RoboDK station: Deployability.rdk

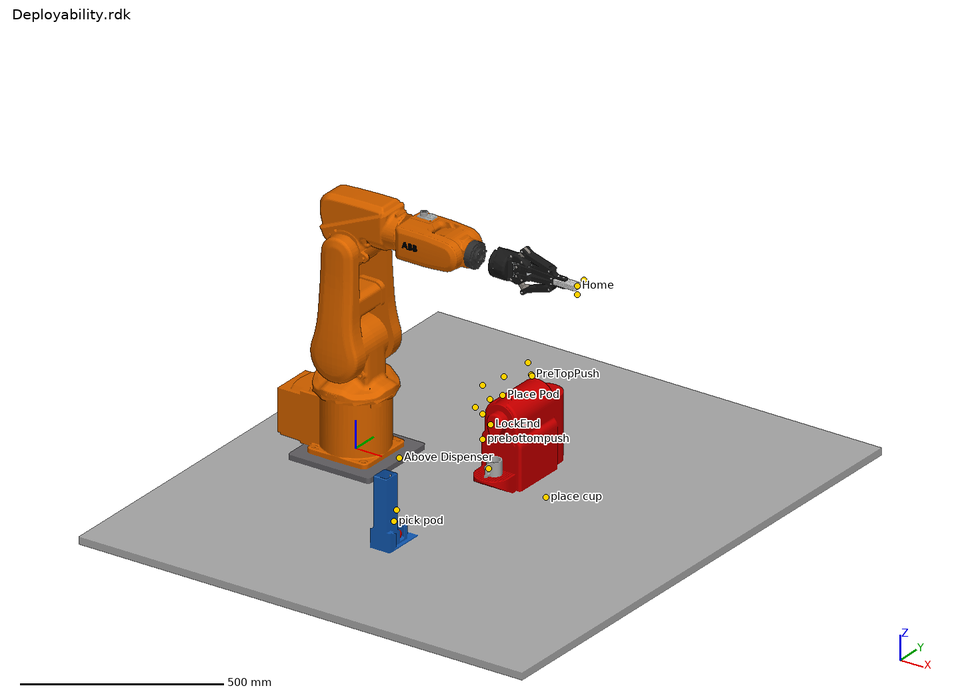
[picture v0: the station drawn from its stored meshes, robots at their saved joint values, targets as dots, program paths as lines]
Station Deployability (saved by RoboDK 5.6.7). Poses are relative to the parent item; angles as X-Y-Z fixed-axis rotations.
Station parameters (name, value as stored): LIN64
  - frame ABB IRB 120-3/0.6 Base at (-2.05, 0, 0) mm
    - target pick pod (Cartesian target) at (354.6, -342.93, 36.52) mm, rotated rx 177.2 ry -1.29 rz 4.29 deg; joints [-43.236, 48.573, -23.215, 1.337, 64.052, 131.893]
    - target Home (Cartesian target) at (664, 0, 630) mm, rotated rx 0 ry 90 rz 0 deg; joints [0, 0, 0, 0, 0, 0]
    - target Place Pod (Cartesian target) at (394.38, 64.87, 228.85) mm, rotated rx 178.74 ry -0.46 rz 90.36 deg; joints [16.786, 24.373, -22.849, 0.084, 87.136, 192.491]
    - target Above Dispenser (Cartesian target) at (372.26, -344.62, 215.16) mm, rotated rx -179.63 ry -1.29 rz 4.29 deg; joints [-43.653, 58.022, -72.664, 1.244, 104.052, 132.364]
    - robot ABB IRB 120-3/0.6: 6 axes, payload 3 kg, reach 580 mm, repeatability 0.01 mm, weight 25 kg
        modified DH rows (alpha deg, a mm, theta deg, d mm): 0, 0, 0, 290; -90, 0, -90, 0; 0, 270, 0, 0; -90, 70, 0, 302; 90, 0, 0, 0; -90, 0, 180, 72
        joint limits [-165, -110, -90, -160, -120, -400] to [165, 110, 70, 160, 120, 400]; home [0, 0, 0, 0, 0, 0]; saved at [-0.052, 0.172, -0.115, 0.095, 0.169, -0.086]
      - tool RobotiQ 2F-140 Gripper (Closed), TCP at (0, 0, 290) mm, size 124 x 75 x 244.3 mm
    - target PreTopPush (Cartesian target) at (397.09, 185.15, 238.21) mm, rotated rx -179.43 ry 2.35 rz -179.98 deg; joints [26.28, 27.432, -27.478, -1.552, 88.195, 26.292] of ABB IRB 120-3/0.6
    - target prebottompush (Cartesian target) at (368.51, 16.26, 120.96) mm, rotated rx 0 ry 90 rz 52.6 deg; joints [-61.285, 60.722, 28.546, -113.883, -90.297, 0.67] of ABB IRB 120-3/0.6
    - target PostTopPush (Cartesian target) at (396.91, -54.26, 245.05) mm, rotated rx -179.43 ry 2.35 rz -179.98 deg; joints [-7.551, 17.486, -15.446, -0.259, 85.559, -7.548] of ABB IRB 120-3/0.6
    - target postbottompush (Cartesian target) at (368.51, 16.26, 269.43) mm, rotated rx 0 ry 90 rz 52.6 deg; joints [-61.285, 29.625, 38.856, -112.389, -98.541, 19.825] of ABB IRB 120-3/0.6
    - target ButtonPush (Cartesian target) at (384.45, 206.23, 222.68) mm, rotated rx 180 ry 13.56 rz 180 deg; joints [34.546, 11.608, -2.276, -8.156, 69.621, 36.65] of ABB IRB 120-3/0.6
    - target LockStart (Cartesian target) at (392.28, 13.5, 239.44) mm, rotated rx -180 ry 1.2 rz 180 deg; joints [2.011, 17.132, -13.99, -0.042, 85.656, 2.013] of ABB IRB 120-3/0.6
    - target LockEnd (Cartesian target) at (393.73, 13.5, 170.14) mm, rotated rx -180 ry 1.2 rz 180 deg; joints [2.003, 16.53, -0.377, -0.044, 72.646, 2.016] of ABB IRB 120-3/0.6
    - target Flex (Cartesian target) at (664, 0, 606.65) mm, rotated rx 0 ry 90 rz 0 deg; joints [0, -0.949, 5.338, 0, -4.389, 0] of ABB IRB 120-3/0.6
    - target Above Pod (Cartesian target) at (360.84, -340.13, 67.96) mm, rotated rx -179.36 ry 1.54 rz 0.85 deg; joints [-42.867, 47.377, -26.349, -0.639, 70.527, 136.515] of ABB IRB 120-3/0.6
    - target Above Drop (Cartesian target) at (398.24, 65.81, 282.08) mm, rotated rx -178.43 ry -0.57 rz 88.39 deg; joints [8.63, 27.474, -36.074, 0.854, 100.039, 100.373] of ABB IRB 120-3/0.6
    - target pre pre toppush (Cartesian target) at (416.98, 380.78, 425.76) mm, rotated rx 169.7 ry 85.71 rz 169.79 deg; joints [81.623, 19.093, 11.361, -90.649, 80.541, 120.963] of ABB IRB 120-3/0.6
    - target Lock Machine (Cartesian target) at (368.51, 16.26, 190.38) mm, rotated rx 0 ry 90 rz 52.6 deg; joints [-61.285, 45.862, 35.295, 66.368, 93.569, -171.904] of ABB IRB 120-3/0.6
    - target pre button (Cartesian target) at (371.56, 206.23, 256.86) mm, rotated rx 180 ry 13.56 rz 180 deg; joints [35.731, 10.177, -6.972, -8.119, 75.853, 36.963] of ABB IRB 120-3/0.6
    - target pick cup (Cartesian target) at (399.81, -3.38, 58.34) mm, rotated rx 136.05 ry 7.69 rz 179.02 deg; joints [-35.158, 42.688, 4.028, 41.312, 72.135, -60.777] of ABB IRB 120-3/0.6
    - target place cup (Cartesian target) at (557.53, 19.04, 14.02) mm, rotated rx 136.05 ry 7.69 rz 179.02 deg; joints [-24.073, 79.25, -53.516, 43.109, 81.693, -39.542] of ABB IRB 120-3/0.6
  - object Tazza_VIP_Mauri at (290, 140, 32) mm, rotated rx 0 ry 0 rz -90 deg, size 60.1 x 40.1 x 39.3 mm, geometry from Tazza_VIP_Mauri.stl
  - object mount at (122.5, 122.5, -15) mm, rotated rx 90 ry 0 rz -90 deg, size 245 x 15 x 245 mm, geometry from mount.STL
  - program Flex Test (4 instructions, listed below)
  - program Gripper Test (6 instructions, listed below)
  - object Base Plate at (-295, -770, -35) mm, rotated rx 90 ry 0 rz 90 deg, size 1540 x 20 x 1330 mm, geometry from Base Plate.STL
  - program Prog3 (1 instructions, listed below)
  - object Body at (386.57, -290, -15) mm, rotated rx 0 ry 0 rz 180 deg, size 68.8 x 120 x 200 mm, geometry from Body.stl
  - object Nsprsocps at (345, -345, 5) mm, rotated rx 0 ry 90 rz 0 deg, size 29.2 x 37.4 x 37.4 mm, geometry from Nsprsocps.stl
  - program Prog5 (4 instructions, listed below)
  - Python program Flex (listed below)
  - object Nespresso Inissia no handle at (332, -25, -15) mm, size 120 x 317.5 x 230 mm, geometry from Nespresso Inissia no handle.STL

--- program Flex Test ---
  Set Ref.: Frame 3 at (-455.88, 959.54, 600.03) mm, rotated rx 88.8 ry 4.28 rz -4.88 deg
  MoveJ (Home) [its target is no longer in the station]
  MoveJ (Flex) [its target is no longer in the station]
  MoveJ (Home) [its target is no longer in the station]

--- program Gripper Test ---
  Set Ref.: Frame 3 at (-455.88, 959.54, 600.03) mm, rotated rx 88.8 ry 4.28 rz -4.88 deg
  Set Tool: RobotiQ 2F-140 Gripper (Closed) at (0, 0, 290) mm
  MoveJ (Home) [its target is no longer in the station]
  Run GripperTesting
  Pause 20.0 s
  MoveJ (Flex) [its target is no longer in the station]

--- program Prog3 (robot ABB IRB 120-3/0.6) ---
  Detach from RobotiQ 2F-140 Gripper (Closed)

--- program Prog5 (robot ABB IRB 120-3/0.6) ---
  Set Ref.: ABB IRB 120-3/0.6 Base
  Set Tool: RobotiQ 2F-140 Gripper (Closed)
  MoveJ (Home)
  Call Flex

--- Python program Flex ---
from robodk.robolink import *

RDK=Robolink()
robot=RDK.Item("ABB IRB 120-3/0.6")

target=RDK.Item("Flex")
robot.MoveJ(target)
